TYPE ST_2DPoint :
STRUCT
	x: LREAL;
	y: LREAL;
END_STRUCT
END_TYPE

(* stored: Version 1.1.0.1, ProductVersion 3.1.4024.3
   DUT ST_2DPoint: Id {893269f3-a8b3-4e7f-b4b8-1a6a52114bcb} *)
